GLOBALCONSTANTS SubStrings (* Global constants *)
  (* Standard: 61499-1 *)
  (* Version 1.0, 2026-08-28, Franz Höpfinger, Meisterschulen am Ostbahnhof *)
  PACKAGE Meins::InputOutputTester::Button_PWM_OPC_UA;
  VAR_GLOBAL CONSTANT
    I1_WRITE : WSTRING := "opc_ua[WRITE;/Objects/DigitalInput/I1,1:s=I1]";
    I2_WRITE : WSTRING := "opc_ua[WRITE;/Objects/DigitalInput/I2,1:s=I2]";
    I3_WRITE : WSTRING := "opc_ua[WRITE;/Objects/DigitalInput/I3,1:s=I3]";
    I4_WRITE : WSTRING := "opc_ua[WRITE;/Objects/DigitalInput/I4,1:s=I4]";
    I5_WRITE : WSTRING := "opc_ua[WRITE;/Objects/DigitalInput/I5,1:s=I5]";
    I6_WRITE : WSTRING := "opc_ua[WRITE;/Objects/DigitalInput/I6,1:s=I6]";
    I7_WRITE : WSTRING := "opc_ua[WRITE;/Objects/DigitalInput/I7,1:s=I7]";
    I8_WRITE : WSTRING := "opc_ua[WRITE;/Objects/DigitalInput/I8,1:s=I8]";
    PWM_Q01_READ : WSTRING := "opc_ua[READ;/Objects/PWM/PWM_Q01,1:s=PWM_Q01]";
    PWM_Q01_WRITE : WSTRING := "opc_ua[WRITE;/Objects/PWM/PWM_Q01,1:s=PWM_Q01]";
    PWM_Q01_SWITCH_READ : WSTRING := "opc_ua[READ;/Objects/PWM/PWM_Q01_SWITCH,1:s=PWM_Q01_SWITCH]";
    PWM_Q01_SWITCH_WRITE : WSTRING := "opc_ua[WRITE;/Objects/PWM/PWM_Q01_SWITCH,1:s=PWM_Q01_SWITCH]";
    PWM_Q01_STATUS_WRITE : WSTRING := "opc_ua[WRITE;/Objects/PWM/PWM_Q01_STATUS,1:s=PWM_Q01_STATUS]";
    PWM_Q02_READ : WSTRING := "opc_ua[READ;/Objects/PWM/PWM_Q02,1:s=PWM_Q02]";
    PWM_Q02_WRITE : WSTRING := "opc_ua[WRITE;/Objects/PWM/PWM_Q02,1:s=PWM_Q02]";
    PWM_Q02_SWITCH_READ : WSTRING := "opc_ua[READ;/Objects/PWM/PWM_Q02_SWITCH,1:s=PWM_Q02_SWITCH]";
    PWM_Q02_SWITCH_WRITE : WSTRING := "opc_ua[WRITE;/Objects/PWM/PWM_Q02_SWITCH,1:s=PWM_Q02_SWITCH]";
    PWM_Q02_STATUS_WRITE : WSTRING := "opc_ua[WRITE;/Objects/PWM/PWM_Q02_STATUS,1:s=PWM_Q02_STATUS]";
    PWM_Q03_READ : WSTRING := "opc_ua[READ;/Objects/PWM/PWM_Q03,1:s=PWM_Q03]";
    PWM_Q03_WRITE : WSTRING := "opc_ua[WRITE;/Objects/PWM/PWM_Q03,1:s=PWM_Q03]";
    PWM_Q03_SWITCH_READ : WSTRING := "opc_ua[READ;/Objects/PWM/PWM_Q03_SWITCH,1:s=PWM_Q03_SWITCH]";
    PWM_Q03_SWITCH_WRITE : WSTRING := "opc_ua[WRITE;/Objects/PWM/PWM_Q03_SWITCH,1:s=PWM_Q03_SWITCH]";
    PWM_Q03_STATUS_WRITE : WSTRING := "opc_ua[WRITE;/Objects/PWM/PWM_Q03_STATUS,1:s=PWM_Q03_STATUS]";
    PWM_Q04_READ : WSTRING := "opc_ua[READ;/Objects/PWM/PWM_Q04,1:s=PWM_Q04]";
    PWM_Q04_WRITE : WSTRING := "opc_ua[WRITE;/Objects/PWM/PWM_Q04,1:s=PWM_Q04]";
    PWM_Q04_SWITCH_READ : WSTRING := "opc_ua[READ;/Objects/PWM/PWM_Q04_SWITCH,1:s=PWM_Q04_SWITCH]";
    PWM_Q04_SWITCH_WRITE : WSTRING := "opc_ua[WRITE;/Objects/PWM/PWM_Q04_SWITCH,1:s=PWM_Q04_SWITCH]";
    PWM_Q04_STATUS_WRITE : WSTRING := "opc_ua[WRITE;/Objects/PWM/PWM_Q04_STATUS,1:s=PWM_Q04_STATUS]";
    PWM_Q05_READ : WSTRING := "opc_ua[READ;/Objects/PWM/PWM_Q05,1:s=PWM_Q05]";
    PWM_Q05_WRITE : WSTRING := "opc_ua[WRITE;/Objects/PWM/PWM_Q05,1:s=PWM_Q05]";
    PWM_Q05_SWITCH_READ : WSTRING := "opc_ua[READ;/Objects/PWM/PWM_Q05_SWITCH,1:s=PWM_Q05_SWITCH]";
    PWM_Q05_SWITCH_WRITE : WSTRING := "opc_ua[WRITE;/Objects/PWM/PWM_Q05_SWITCH,1:s=PWM_Q05_SWITCH]";
    PWM_Q05_STATUS_WRITE : WSTRING := "opc_ua[WRITE;/Objects/PWM/PWM_Q05_STATUS,1:s=PWM_Q05_STATUS]";
    PWM_Q06_READ : WSTRING := "opc_ua[READ;/Objects/PWM/PWM_Q06,1:s=PWM_Q06]";
    PWM_Q06_WRITE : WSTRING := "opc_ua[WRITE;/Objects/PWM/PWM_Q06,1:s=PWM_Q06]";
    PWM_Q06_SWITCH_READ : WSTRING := "opc_ua[READ;/Objects/PWM/PWM_Q06_SWITCH,1:s=PWM_Q06_SWITCH]";
    PWM_Q06_SWITCH_WRITE : WSTRING := "opc_ua[WRITE;/Objects/PWM/PWM_Q06_SWITCH,1:s=PWM_Q06_SWITCH]";
    PWM_Q06_STATUS_WRITE : WSTRING := "opc_ua[WRITE;/Objects/PWM/PWM_Q06_STATUS,1:s=PWM_Q06_STATUS]";
    PWM_Q07_READ : WSTRING := "opc_ua[READ;/Objects/PWM/PWM_Q07,1:s=PWM_Q07]";
    PWM_Q07_WRITE : WSTRING := "opc_ua[WRITE;/Objects/PWM/PWM_Q07,1:s=PWM_Q07]";
    PWM_Q07_SWITCH_READ : WSTRING := "opc_ua[READ;/Objects/PWM/PWM_Q07_SWITCH,1:s=PWM_Q07_SWITCH]";
    PWM_Q07_SWITCH_WRITE : WSTRING := "opc_ua[WRITE;/Objects/PWM/PWM_Q07_SWITCH,1:s=PWM_Q07_SWITCH]";
    PWM_Q07_STATUS_WRITE : WSTRING := "opc_ua[WRITE;/Objects/PWM/PWM_Q07_STATUS,1:s=PWM_Q07_STATUS]";
    PWM_Q08_READ : WSTRING := "opc_ua[READ;/Objects/PWM/PWM_Q08,1:s=PWM_Q08]";
    PWM_Q08_WRITE : WSTRING := "opc_ua[WRITE;/Objects/PWM/PWM_Q08,1:s=PWM_Q08]";
    PWM_Q08_SWITCH_READ : WSTRING := "opc_ua[READ;/Objects/PWM/PWM_Q08_SWITCH,1:s=PWM_Q08_SWITCH]";
    PWM_Q08_SWITCH_WRITE : WSTRING := "opc_ua[WRITE;/Objects/PWM/PWM_Q08_SWITCH,1:s=PWM_Q08_SWITCH]";
    PWM_Q08_STATUS_WRITE : WSTRING := "opc_ua[WRITE;/Objects/PWM/PWM_Q08_STATUS,1:s=PWM_Q08_STATUS]";
    PWM_Q09_READ : WSTRING := "opc_ua[READ;/Objects/PWM/PWM_Q09,1:s=PWM_Q09]";
    PWM_Q09_WRITE : WSTRING := "opc_ua[WRITE;/Objects/PWM/PWM_Q09,1:s=PWM_Q09]";
    PWM_Q09_SWITCH_READ : WSTRING := "opc_ua[READ;/Objects/PWM/PWM_Q09_SWITCH,1:s=PWM_Q09_SWITCH]";
    PWM_Q09_SWITCH_WRITE : WSTRING := "opc_ua[WRITE;/Objects/PWM/PWM_Q09_SWITCH,1:s=PWM_Q09_SWITCH]";
    PWM_Q09_STATUS_WRITE : WSTRING := "opc_ua[WRITE;/Objects/PWM/PWM_Q09_STATUS,1:s=PWM_Q09_STATUS]";
    PWM_Q10_READ : WSTRING := "opc_ua[READ;/Objects/PWM/PWM_Q10,1:s=PWM_Q10]";
    PWM_Q10_WRITE : WSTRING := "opc_ua[WRITE;/Objects/PWM/PWM_Q10,1:s=PWM_Q10]";
    PWM_Q10_SWITCH_READ : WSTRING := "opc_ua[READ;/Objects/PWM/PWM_Q10_SWITCH,1:s=PWM_Q10_SWITCH]";
    PWM_Q10_SWITCH_WRITE : WSTRING := "opc_ua[WRITE;/Objects/PWM/PWM_Q10_SWITCH,1:s=PWM_Q10_SWITCH]";
    PWM_Q10_STATUS_WRITE : WSTRING := "opc_ua[WRITE;/Objects/PWM/PWM_Q10_STATUS,1:s=PWM_Q10_STATUS]";
    PWM_Q11_READ : WSTRING := "opc_ua[READ;/Objects/PWM/PWM_Q11,1:s=PWM_Q11]";
    PWM_Q11_WRITE : WSTRING := "opc_ua[WRITE;/Objects/PWM/PWM_Q11,1:s=PWM_Q11]";
    PWM_Q11_SWITCH_READ : WSTRING := "opc_ua[READ;/Objects/PWM/PWM_Q11_SWITCH,1:s=PWM_Q11_SWITCH]";
    PWM_Q11_SWITCH_WRITE : WSTRING := "opc_ua[WRITE;/Objects/PWM/PWM_Q11_SWITCH,1:s=PWM_Q11_SWITCH]";
    PWM_Q11_STATUS_WRITE : WSTRING := "opc_ua[WRITE;/Objects/PWM/PWM_Q11_STATUS,1:s=PWM_Q11_STATUS]";
    PWM_Q12_READ : WSTRING := "opc_ua[READ;/Objects/PWM/PWM_Q12,1:s=PWM_Q12]";
    PWM_Q12_WRITE : WSTRING := "opc_ua[WRITE;/Objects/PWM/PWM_Q12,1:s=PWM_Q12]";
    PWM_Q12_SWITCH_READ : WSTRING := "opc_ua[READ;/Objects/PWM/PWM_Q12_SWITCH,1:s=PWM_Q12_SWITCH]";
    PWM_Q12_SWITCH_WRITE : WSTRING := "opc_ua[WRITE;/Objects/PWM/PWM_Q12_SWITCH,1:s=PWM_Q12_SWITCH]";
    PWM_Q12_STATUS_WRITE : WSTRING := "opc_ua[WRITE;/Objects/PWM/PWM_Q12_STATUS,1:s=PWM_Q12_STATUS]";
    Tick_WRITE : WSTRING := "opc_ua[WRITE;/Objects/System/Tick,1:s=System.Tick]";
  END_VAR
END_GLOBALCONSTANTS
